PROGRAM Comp01_Devices
VAR
	Step_0: Step;
END_VAR

Actuators();
Servos();

ACTION Actuators:
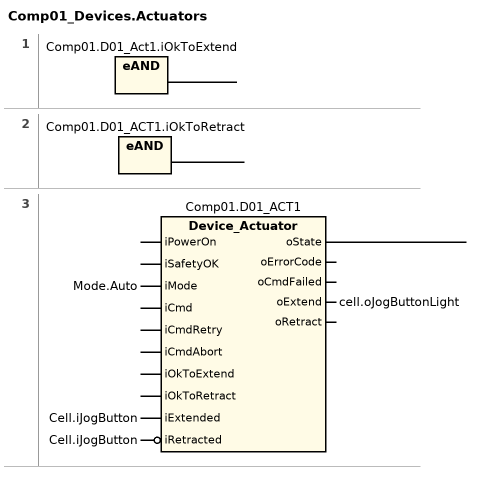
// NETWORK 1
Comp01.D01_Act1.iOkToExtend(); // eAND

// NETWORK 2
Comp01.D01_ACT1.iOkToRetract(); // eAND

// NETWORK 3
Comp01.D01_ACT1(
    iMode := Mode.Auto,
    iExtended := Cell.iJogButton,
    iRetracted := NOT Cell.iJogButton,
    oExtend => cell.oJogButtonLight); // Device_Actuator
END_ACTION

ACTION Servos:
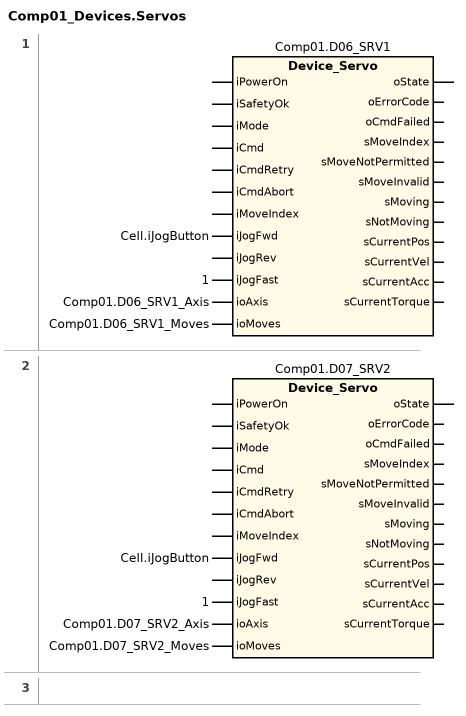
// NETWORK 1
Comp01.D06_SRV1(
    iJogFwd := Cell.iJogButton,
    iJogFast := 1,
    ioAxis := Comp01.D06_SRV1_Axis,
    ioMoves := Comp01.D06_SRV1_Moves); // Device_Servo

// NETWORK 2
Comp01.D07_SRV2(
    iJogFwd := Cell.iJogButton,
    iJogFast := 1,
    ioAxis := Comp01.D07_SRV2_Axis,
    ioMoves := Comp01.D07_SRV2_Moves); // Device_Servo

// NETWORK 3
END_ACTION

END_PROGRAM

(* stored: Version 1.1.0.1, ProductVersion 3.1.4022.11
   POU Comp01_Devices: Id {f0a046c5-ec80-4bdc-848e-27d048afa24d}, SpecialFunc None
   Action Actuators: Id {6d8a1d68-4091-4119-9dcf-9feebf32806f}
   Action Servos: Id {dfa8bfe5-7073-4b59-a3cb-a32e24979de3} *)
